% RSLogix 500 project DRYER MCM NOVEMBER NEW ZELAND 1-7-2018 CURRENT_JEFF_EMAIL_TO_EULISES.RSS, saved by version 11.00.00.00 %
PROJECT "ML1200"    % processor: MicroLogix 1200; MAIN_PROG %

PROGRAM FILES
  LAD 2 "MAIN_PROG"  11 rungs
  LAD 3 "DRYER CONT"  11 rungs
  LAD 4 "TEMPERATUR"  32 rungs
  LAD 5 "AIR PRES."  7 rungs
  LAD 6 "HUMIDITY"  13 rungs
  LAD 7 "RHL-TEMP"  2 rungs  % HEATING CONTROLS %
  LAD 8 "HEAT CONTR"  39 rungs
  LAD 9 "HOUR METER"  6 rungs
  LAD 10 "CONV CLEAN"  18 rungs  % Brush Cleaning %
  LAD 11 "FAULTS"  8 rungs

DATA FILES
  O0 OUTPUT  8 elements
  I1 INPUT  19 elements
  S2 STATUS  66 elements
  B3 BINARY  6 elements
  T4 TIMER  11 elements
  C5 COUNTER  1 elements
  R6 CONTROL  1 elements
  N7 INTEGER  80 elements
  F8 FLOAT  1 elements
  PD9 DRYER  4 elements

LADDER 2 "MAIN_PROG"
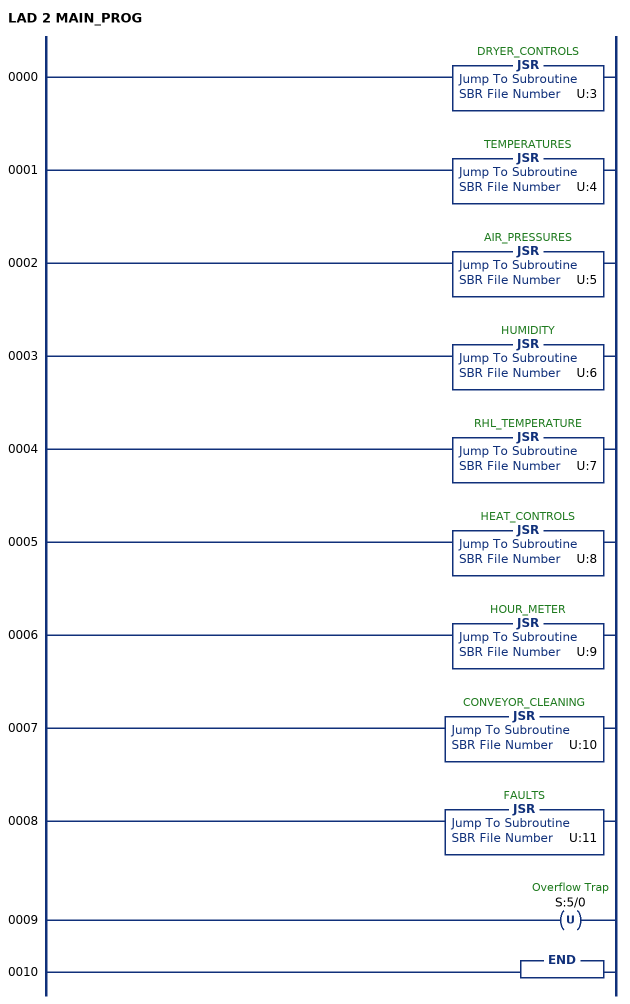
% Rung: 0 %
SOR JSR U:3 EOR
%   U:3  DRYER_CONTROLS %
% Rung: 1 %
SOR JSR U:4 EOR
%   U:4  TEMPERATURES %
% Rung: 2 %
SOR JSR U:5 EOR
%   U:5  AIR_PRESSURES %
% Rung: 3 %
SOR JSR U:6 EOR
%   U:6  HUMIDITY %
% Rung: 4 %
SOR JSR U:7 EOR
%   U:7  RHL_TEMPERATURE %
% Rung: 5 %
SOR JSR U:8 EOR
%   U:8  HEAT_CONTROLS %
% Rung: 6 %
SOR JSR U:9 EOR
%   U:9  HOUR_METER %
% Rung: 7 %
SOR JSR U:10 EOR
%   U:10  CONVEYOR_CLEANING %
% Rung: 8 %
SOR JSR U:11 EOR
%   U:11  FAULTS %
% Rung: 9 %
SOR OTU S:5/0 EOR
%   S:5/0  "Overflow Trap" %
% Rung: 10 %
SOR END EOR

LADDER 3 "DRYER CONT"
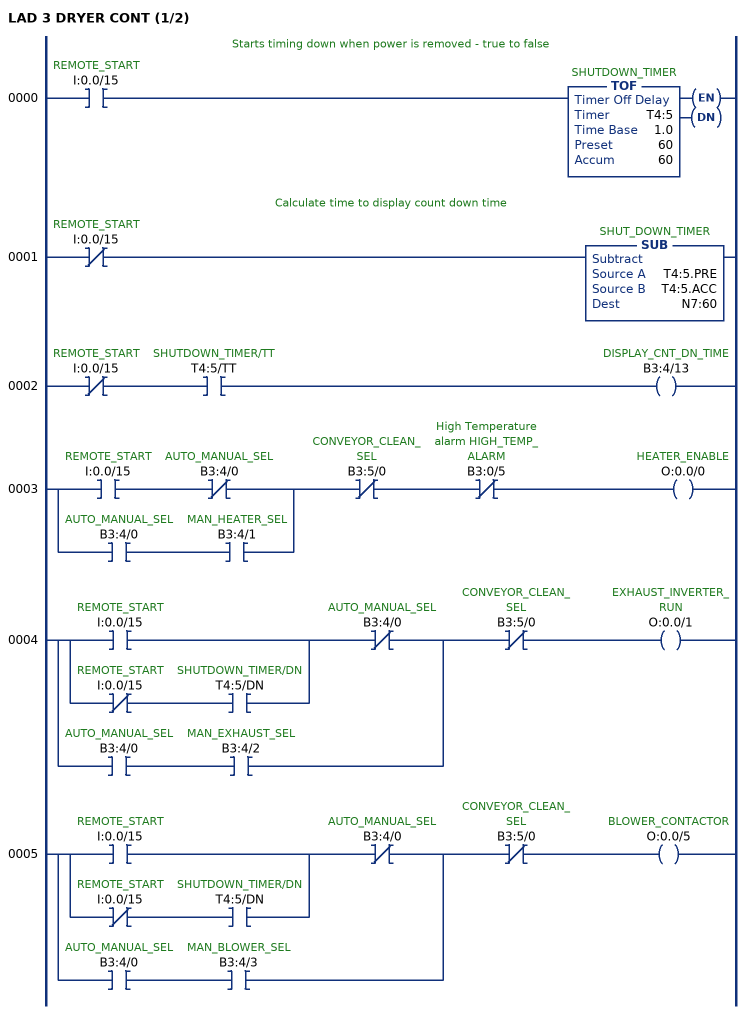
% Rung: 0 %
% Starts timing down when power is removed - true to false %
SOR XIC I:0.0/15 TOF T4:5 1.0 60 60 EOR
%   I:0.0/15  REMOTE_START %
%   T4:5  SHUTDOWN_TIMER %
% Rung: 1 %
% Calculate time to display count down time %
SOR XIO I:0.0/15 SUB T4:5.PRE T4:5.ACC N7:60 EOR
%   I:0.0/15  REMOTE_START %
%   T4:5  SHUTDOWN_TIMER %
%   N7:60  SHUT_DOWN_TIMER %
% Rung: 2 %
SOR XIO I:0.0/15 XIC T4:5/TT OTE B3:4/13 EOR
%   I:0.0/15  REMOTE_START %
%   T4:5  SHUTDOWN_TIMER %
%   B3:4/13  DISPLAY_CNT_DN_TIME %
% Rung: 3 %
SOR BST XIC I:0.0/15 XIO B3:4/0 NXB XIC B3:4/0 XIC B3:4/1 BND XIO B3:5/0 XIO B3:0/5 OTE O:0.0/0 EOR
%   I:0.0/15  REMOTE_START %
%   B3:4/0  AUTO_MANUAL_SEL %
%   B3:4/1  MAN_HEATER_SEL %
%   B3:5/0  CONVEYOR_CLEAN_SEL %
%   B3:0/5  HIGH_TEMP_ALARM  "High Temperature alarm" %
%   O:0.0/0  HEATER_ENABLE %
% Rung: 4 %
SOR BST BST XIC I:0.0/15 NXB XIO I:0.0/15 XIC T4:5/DN BND XIO B3:4/0 NXB XIC B3:4/0 XIC B3:4/2 BND XIO B3:5/0 OTE O:0.0/1 EOR
%   I:0.0/15  REMOTE_START %
%   T4:5  SHUTDOWN_TIMER %
%   B3:4/0  AUTO_MANUAL_SEL %
%   B3:4/2  MAN_EXHAUST_SEL %
%   B3:5/0  CONVEYOR_CLEAN_SEL %
%   O:0.0/1  EXHAUST_INVERTER_RUN %
% Rung: 5 %
SOR BST BST XIC I:0.0/15 NXB XIO I:0.0/15 XIC T4:5/DN BND XIO B3:4/0 NXB XIC B3:4/0 XIC B3:4/3 BND XIO B3:5/0 OTE O:0.0/5 EOR
%   I:0.0/15  REMOTE_START %
%   T4:5  SHUTDOWN_TIMER %
%   B3:4/0  AUTO_MANUAL_SEL %
%   B3:4/3  MAN_BLOWER_SEL %
%   B3:5/0  CONVEYOR_CLEAN_SEL %
%   O:0.0/5  BLOWER_CONTACTOR %

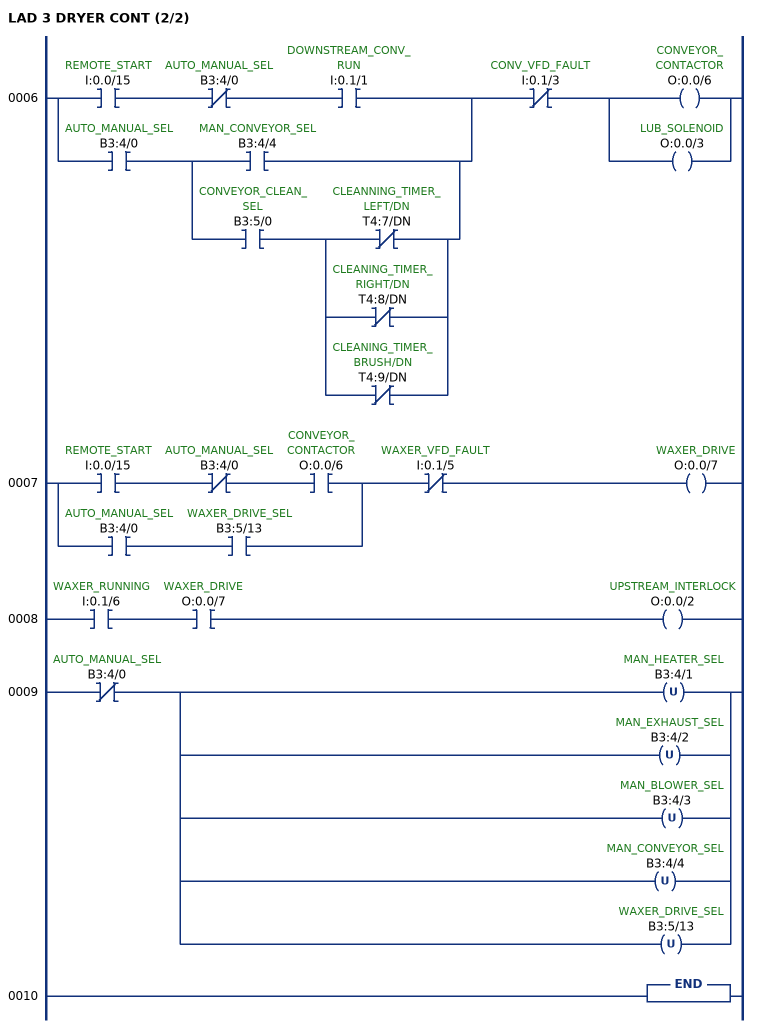
% Rung: 6 %
SOR BST XIC I:0.0/15 XIO B3:4/0 XIC I:0.1/1 NXB XIC B3:4/0 BST XIC B3:4/4 NXB XIC B3:5/0 BST XIO T4:7/DN NXB BST XIO T4:8/DN NXB XIO T4:9/DN BND BND BND BND XIO I:0.1/3 BST OTE O:0.0/6 NXB OTE O:0.0/3 BND EOR
%   I:0.0/15  REMOTE_START %
%   B3:4/0  AUTO_MANUAL_SEL %
%   I:0.1/1  DOWNSTREAM_CONV_RUN %
%   B3:4/4  MAN_CONVEYOR_SEL %
%   B3:5/0  CONVEYOR_CLEAN_SEL %
%   T4:7  CLEANNING_TIMER_LEFT %
%   T4:8  CLEANING_TIMER_RIGHT %
%   T4:9  CLEANING_TIMER_BRUSH %
%   I:0.1/3  CONV_VFD_FAULT %
%   O:0.0/6  CONVEYOR_CONTACTOR %
%   O:0.0/3  LUB_SOLENOID %
% Rung: 7 %
SOR BST XIC I:0.0/15 XIO B3:4/0 XIC O:0.0/6 NXB XIC B3:4/0 XIC B3:5/13 BND XIO I:0.1/5 OTE O:0.0/7 EOR
%   I:0.0/15  REMOTE_START %
%   B3:4/0  AUTO_MANUAL_SEL %
%   O:0.0/6  CONVEYOR_CONTACTOR %
%   B3:5/13  WAXER_DRIVE_SEL %
%   I:0.1/5  WAXER_VFD_FAULT %
%   O:0.0/7  WAXER_DRIVE %
% Rung: 8 %
SOR XIC I:0.1/6 XIC O:0.0/7 OTE O:0.0/2 EOR
%   I:0.1/6  WAXER_RUNNING %
%   O:0.0/7  WAXER_DRIVE %
%   O:0.0/2  UPSTREAM_INTERLOCK %
% Rung: 9 %
SOR XIO B3:4/0 BST BST BST BST OTU B3:4/1 NXB OTU B3:4/2 BND NXB OTU B3:4/3 BND NXB OTU B3:4/4 BND NXB OTU B3:5/13 BND EOR
%   B3:4/0  AUTO_MANUAL_SEL %
%   B3:4/1  MAN_HEATER_SEL %
%   B3:4/2  MAN_EXHAUST_SEL %
%   B3:4/3  MAN_BLOWER_SEL %
%   B3:4/4  MAN_CONVEYOR_SEL %
%   B3:5/13  WAXER_DRIVE_SEL %
% Rung: 10 %
SOR END EOR

LADDER 4 "TEMPERATUR"
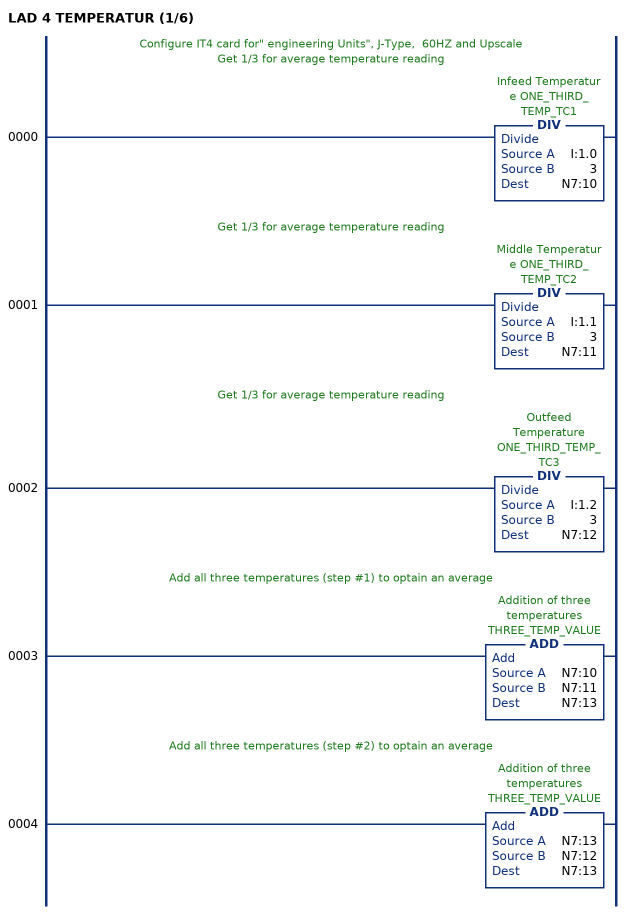
% Rung: 0 %
% Configure IT4 card for" engineering Units", J-Type,  60HZ and Upscale
% Get 1/3 for average temperature reading %
SOR DIV I:1.0 3 N7:10 EOR
%   I:1.0  INFEED_TEMP %
%   N7:10  ONE_THIRD_TEMP_TC1  "Infeed Temperature" %
% Rung: 1 %
% Get 1/3 for average temperature reading %
SOR DIV I:1.1 3 N7:11 EOR
%   I:1.1  MIDDLE_TEMP %
%   N7:11  ONE_THIRD_TEMP_TC2  "Middle Temperature" %
% Rung: 2 %
% Get 1/3 for average temperature reading %
SOR DIV I:1.2 3 N7:12 EOR
%   I:1.2  OUTFEED_TEMP %
%   N7:12  ONE_THIRD_TEMP_TC3  "Outfeed Temperature" %
% Rung: 3 %
% Add all three temperatures (step #1) to optain an average %
SOR ADD N7:10 N7:11 N7:13 EOR
%   N7:10  ONE_THIRD_TEMP_TC1  "Infeed Temperature" %
%   N7:11  ONE_THIRD_TEMP_TC2  "Middle Temperature" %
%   N7:13  THREE_TEMP_VALUE  "Addition of three temperatures" %
% Rung: 4 %
% Add all three temperatures (step #2) to optain an average %
SOR ADD N7:13 N7:12 N7:13 EOR
%   N7:13  THREE_TEMP_VALUE  "Addition of three temperatures" %
%   N7:12  ONE_THIRD_TEMP_TC3  "Outfeed Temperature" %

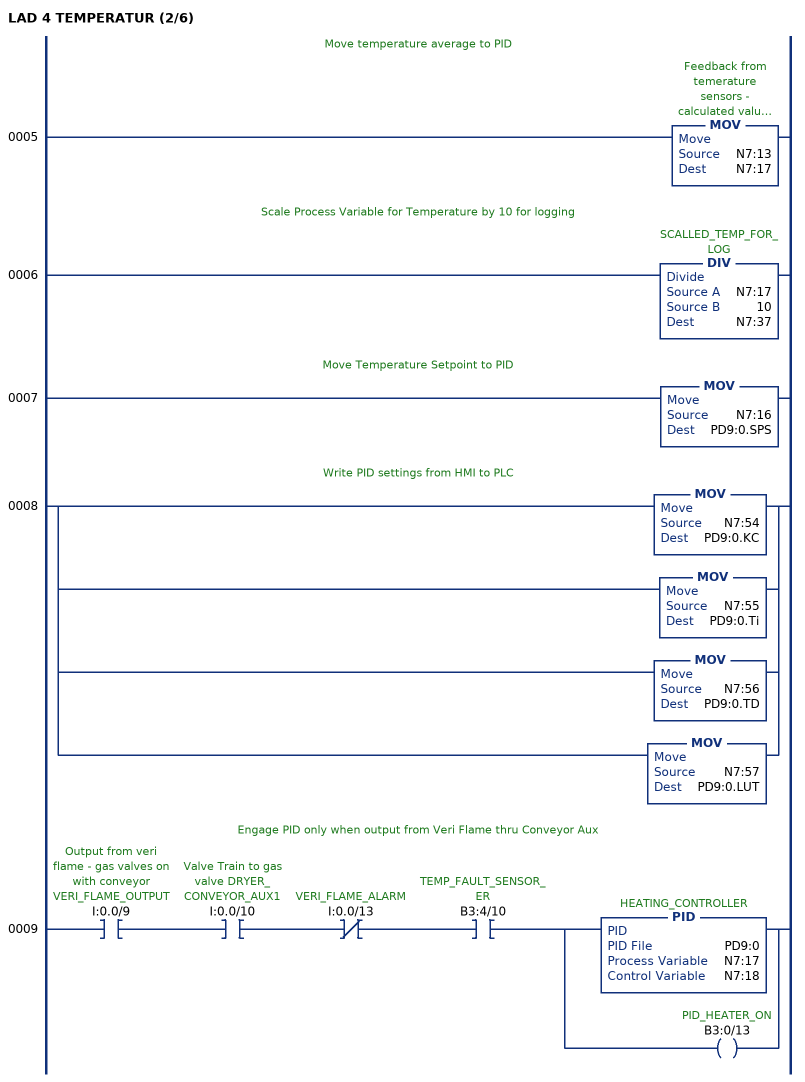
% Rung: 5 %
% Move temperature average to PID %
SOR MOV N7:13 N7:17 EOR
%   N7:13  THREE_TEMP_VALUE  "Addition of three temperatures" %
%   N7:17  PV_TEMP_PROCESS_VAR  "Feedback from temerature sensors - calculated value" %
% Rung: 6 %
% Scale Process Variable for Temperature by 10 for logging %
SOR DIV N7:17 10 N7:37 EOR
%   N7:17  PV_TEMP_PROCESS_VAR  "Feedback from temerature sensors - calculated value" %
%   N7:37  SCALLED_TEMP_FOR_LOG %
% Rung: 7 %
% Move Temperature Setpoint to PID %
SOR MOV N7:16 PD9:0.SPS EOR
%   N7:16  SPS_TEMP_SETPOINT  "Display Input Value - desired Temperature" %
% Rung: 8 %
% Write PID settings from HMI to PLC %
SOR BST BST BST MOV N7:54 PD9:0.KC NXB MOV N7:55 PD9:0.Ti BND NXB MOV N7:56 PD9:0.TD BND NXB MOV N7:57 PD9:0.LUT BND EOR
%   N7:54  PID_KC %
%   N7:55  PID_TI %
%   N7:56  PID_TD %
%   N7:57  PID_LUT %
% Rung: 9 %
% Engage PID only when output from Veri Flame thru Conveyor Aux %
SOR XIC I:0.0/9 XIC I:0.0/10 XIO I:0.0/13 XIC B3:4/10 BST PID PD9:0 N7:17 N7:18 NXB OTE B3:0/13 BND EOR
%   I:0.0/9  VERI_FLAME_OUTPUT  "Output from veri flame - gas valves on with conveyor" %
%   I:0.0/10  DRYER_CONVEYOR_AUX1  "Valve Train to gas valve" %
%   I:0.0/13  VERI_FLAME_ALARM %
%   B3:4/10  TEMP_FAULT_SENSOR_ER %
%   PD9:0  HEATING_CONTROLLER %
%   N7:17  PV_TEMP_PROCESS_VAR  "Feedback from temerature sensors - calculated value" %
%   N7:18  CV_TEMP_CONTROL_VAR  "Output value to output for output card" %
%   B3:0/13  PID_HEATER_ON %

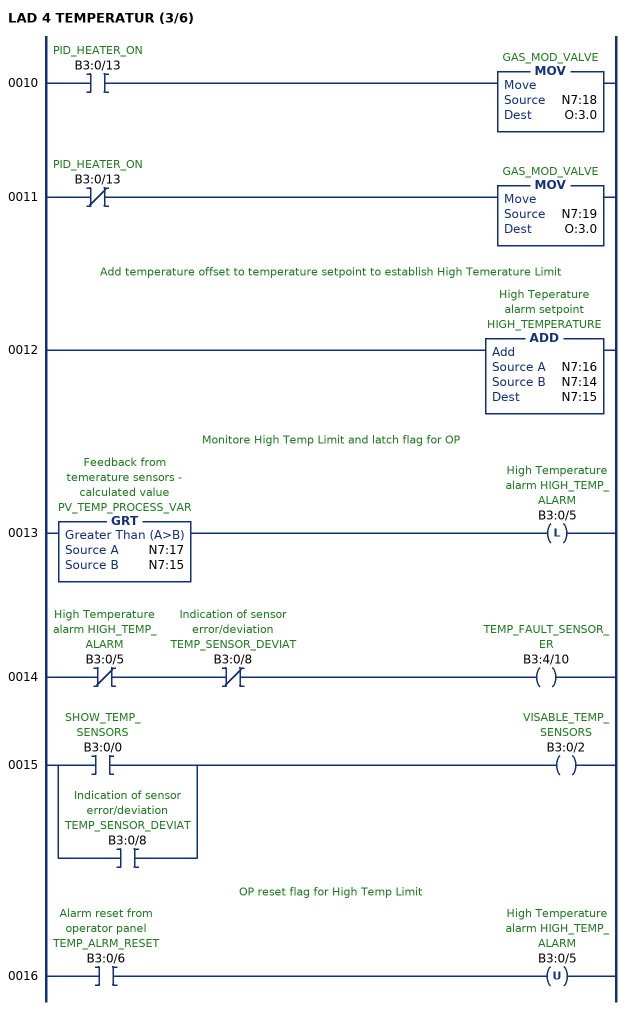
% Rung: 10 %
SOR XIC B3:0/13 MOV N7:18 O:3.0 EOR
%   B3:0/13  PID_HEATER_ON %
%   N7:18  CV_TEMP_CONTROL_VAR  "Output value to output for output card" %
%   O:3.0  GAS_MOD_VALVE %
% Rung: 11 %
SOR XIO B3:0/13 MOV N7:19 O:3.0 EOR
%   B3:0/13  PID_HEATER_ON %
%   N7:19  MIN_GAS_VALVE_POS  "When Conveyor Aux is off, throttle valve back" %
%   O:3.0  GAS_MOD_VALVE %
% Rung: 12 %
% Add temperature offset to temperature setpoint to establish High Temerature Limit %
SOR ADD N7:16 N7:14 N7:15 EOR
%   N7:16  SPS_TEMP_SETPOINT  "Display Input Value - desired Temperature" %
%   N7:14  HIGH_TEMP_OFFSET  "Value added to Temp Setpoint to set high temerature" %
%   N7:15  HIGH_TEMPERATURE  "High Teperature alarm setpoint" %
% Rung: 13 %
% Monitore High Temp Limit and latch flag for OP %
SOR GRT N7:17 N7:15 OTL B3:0/5 EOR
%   N7:17  PV_TEMP_PROCESS_VAR  "Feedback from temerature sensors - calculated value" %
%   N7:15  HIGH_TEMPERATURE  "High Teperature alarm setpoint" %
%   B3:0/5  HIGH_TEMP_ALARM  "High Temperature alarm" %
% Rung: 14 %
SOR XIO B3:0/5 XIO B3:0/8 OTE B3:4/10 EOR
%   B3:0/5  HIGH_TEMP_ALARM  "High Temperature alarm" %
%   B3:0/8  TEMP_SENSOR_DEVIAT  "Indication of sensor error/deviation" %
%   B3:4/10  TEMP_FAULT_SENSOR_ER %
% Rung: 15 %
SOR BST XIC B3:0/0 NXB XIC B3:0/8 BND OTE B3:0/2 EOR
%   B3:0/0  SHOW_TEMP_SENSORS %
%   B3:0/8  TEMP_SENSOR_DEVIAT  "Indication of sensor error/deviation" %
%   B3:0/2  VISABLE_TEMP_SENSORS %
% Rung: 16 %
% OP reset flag for High Temp Limit %
SOR XIC B3:0/6 OTU B3:0/5 EOR
%   B3:0/6  TEMP_ALRM_RESET  "Alarm reset from operator panel" %
%   B3:0/5  HIGH_TEMP_ALARM  "High Temperature alarm" %

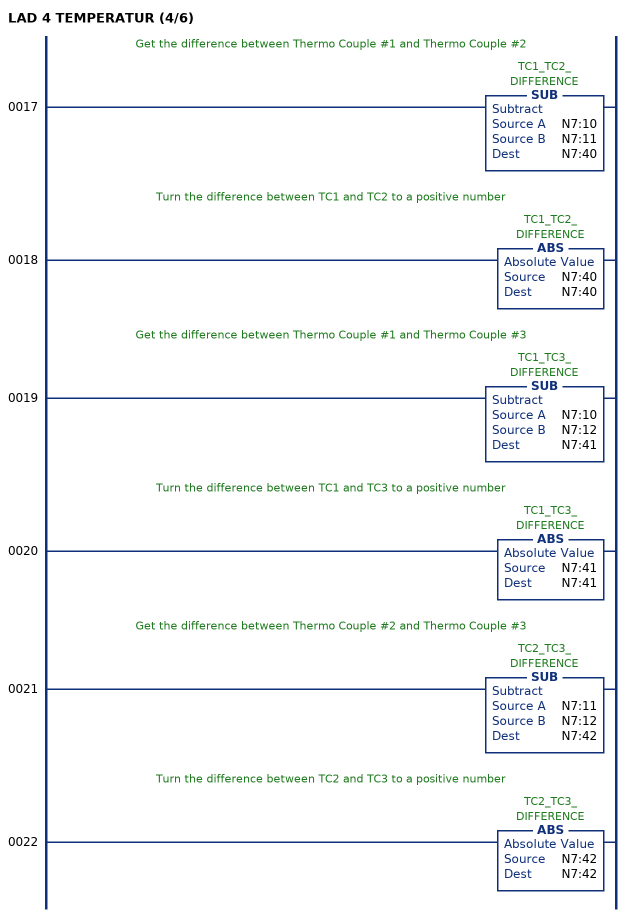
% Rung: 17 %
% Get the difference between Thermo Couple #1 and Thermo Couple #2 %
SOR SUB N7:10 N7:11 N7:40 EOR
%   N7:10  ONE_THIRD_TEMP_TC1  "Infeed Temperature" %
%   N7:11  ONE_THIRD_TEMP_TC2  "Middle Temperature" %
%   N7:40  TC1_TC2_DIFFERENCE %
% Rung: 18 %
% Turn the difference between TC1 and TC2 to a positive number %
SOR ABS N7:40 N7:40 EOR
%   N7:40  TC1_TC2_DIFFERENCE %
% Rung: 19 %
% Get the difference between Thermo Couple #1 and Thermo Couple #3 %
SOR SUB N7:10 N7:12 N7:41 EOR
%   N7:10  ONE_THIRD_TEMP_TC1  "Infeed Temperature" %
%   N7:12  ONE_THIRD_TEMP_TC3  "Outfeed Temperature" %
%   N7:41  TC1_TC3_DIFFERENCE %
% Rung: 20 %
% Turn the difference between TC1 and TC3 to a positive number %
SOR ABS N7:41 N7:41 EOR
%   N7:41  TC1_TC3_DIFFERENCE %
% Rung: 21 %
% Get the difference between Thermo Couple #2 and Thermo Couple #3 %
SOR SUB N7:11 N7:12 N7:42 EOR
%   N7:11  ONE_THIRD_TEMP_TC2  "Middle Temperature" %
%   N7:12  ONE_THIRD_TEMP_TC3  "Outfeed Temperature" %
%   N7:42  TC2_TC3_DIFFERENCE %
% Rung: 22 %
% Turn the difference between TC2 and TC3 to a positive number %
SOR ABS N7:42 N7:42 EOR
%   N7:42  TC2_TC3_DIFFERENCE %

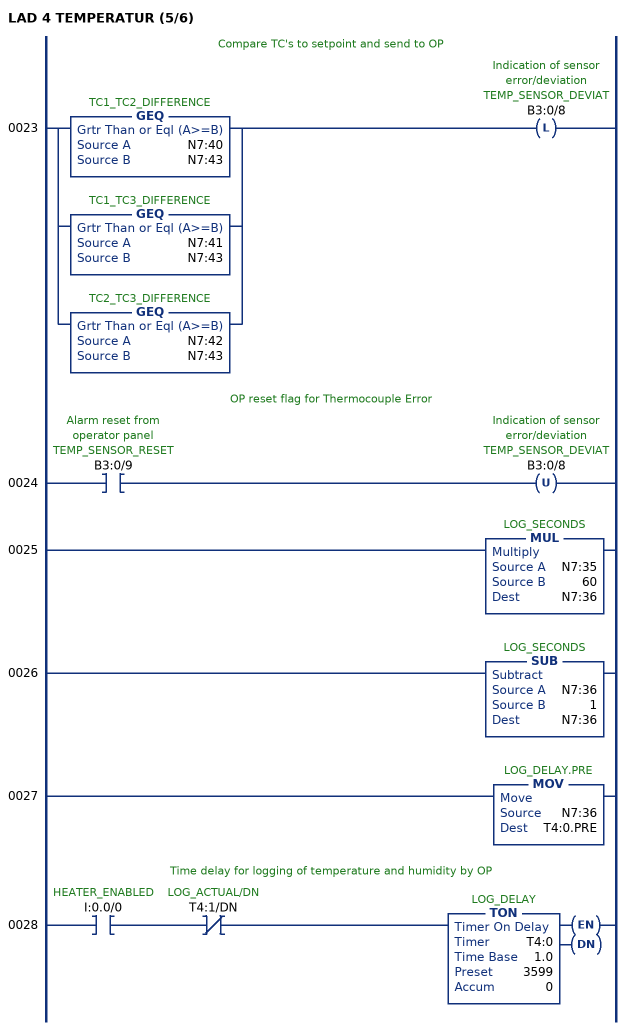
% Rung: 23 %
% Compare TC's to setpoint and send to OP %
SOR BST GEQ N7:40 N7:43 NXB BST GEQ N7:41 N7:43 NXB GEQ N7:42 N7:43 BND BND OTL B3:0/8 EOR
%   N7:40  TC1_TC2_DIFFERENCE %
%   N7:43  MAX_TEMP_SENSOR_DEV %
%   N7:41  TC1_TC3_DIFFERENCE %
%   N7:42  TC2_TC3_DIFFERENCE %
%   B3:0/8  TEMP_SENSOR_DEVIAT  "Indication of sensor error/deviation" %
% Rung: 24 %
% OP reset flag for Thermocouple Error %
SOR XIC B3:0/9 OTU B3:0/8 EOR
%   B3:0/9  TEMP_SENSOR_RESET  "Alarm reset from operator panel" %
%   B3:0/8  TEMP_SENSOR_DEVIAT  "Indication of sensor error/deviation" %
% Rung: 25 %
SOR MUL N7:35 60 N7:36 EOR
%   N7:35  LOG_MINUTES %
%   N7:36  LOG_SECONDS %
% Rung: 26 %
SOR SUB N7:36 1 N7:36 EOR
%   N7:36  LOG_SECONDS %
% Rung: 27 %
SOR MOV N7:36 T4:0.PRE EOR
%   N7:36  LOG_SECONDS %
%   T4:0  LOG_DELAY %
% Rung: 28 %
% Time delay for logging of temperature and humidity by OP %
SOR XIC I:0.0/0 XIO T4:1/DN TON T4:0 1.0 3599 0 EOR
%   I:0.0/0  HEATER_ENABLED %
%   T4:1  LOG_ACTUAL %
%   T4:0  LOG_DELAY %

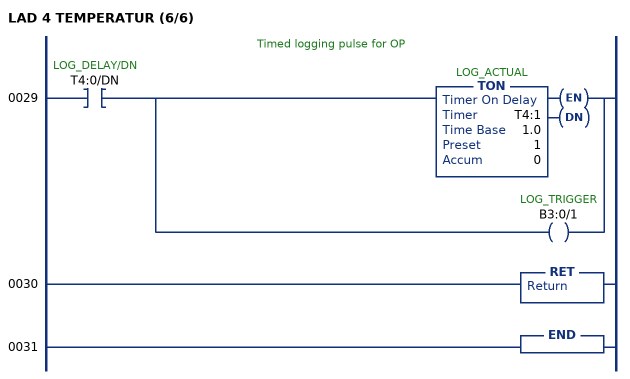
% Rung: 29 %
% Timed logging pulse for OP %
SOR XIC T4:0/DN BST TON T4:1 1.0 1 0 NXB OTE B3:0/1 BND EOR
%   T4:0  LOG_DELAY %
%   T4:1  LOG_ACTUAL %
%   B3:0/1  LOG_TRIGGER %
% Rung: 30 %
SOR RET EOR
% Rung: 31 %
SOR END EOR

LADDER 5 "AIR PRES."
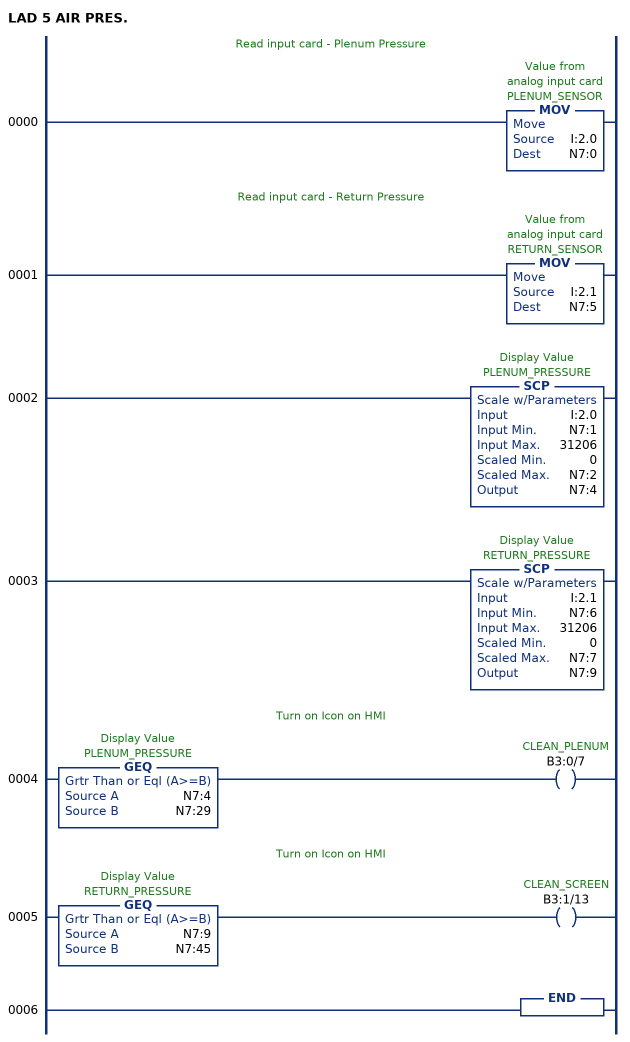
% Rung: 0 %
% Read input card - Plenum Pressure %
SOR MOV I:2.0 N7:0 EOR
%   N7:0  PLENUM_SENSOR  "Value from analog input card" %
% Rung: 1 %
% Read input card - Return Pressure %
SOR MOV I:2.1 N7:5 EOR
%   N7:5  RETURN_SENSOR  "Value from analog input card" %
% Rung: 2 %
SOR SCP I:2.0 N7:1 31206 0 N7:2 N7:4 EOR
%   N7:1  PLENUM_ZERO  "The amount needed to return a zero value with no pressure" %
%   N7:2  PLENUM_SCALLING_MAX  "Max range of sensor" %
%   N7:4  PLENUM_PRESSURE  "Display Value" %
% Rung: 3 %
SOR SCP I:2.1 N7:6 31206 0 N7:7 N7:9 EOR
%   N7:6  RETURN_ZERO  "The amount needed to return a zero value with no pressure" %
%   N7:7  RETURN_SCALING_MAX  "Max range of sensor" %
%   N7:9  RETURN_PRESSURE  "Display Value" %
% Rung: 4 %
% Turn on Icon on HMI %
SOR GEQ N7:4 N7:29 OTE B3:0/7 EOR
%   N7:4  PLENUM_PRESSURE  "Display Value" %
%   N7:29  PLENUM_ALARM  "signal Operator Panel that cleaning is required" %
%   B3:0/7  CLEAN_PLENUM %
% Rung: 5 %
% Turn on Icon on HMI %
SOR GEQ N7:9 N7:45 OTE B3:1/13 EOR
%   N7:9  RETURN_PRESSURE  "Display Value" %
%   N7:45  CLEAN_SCREEN_ALARM %
%   B3:1/13  CLEAN_SCREEN %
% Rung: 6 %
SOR END EOR

LADDER 6 "HUMIDITY"
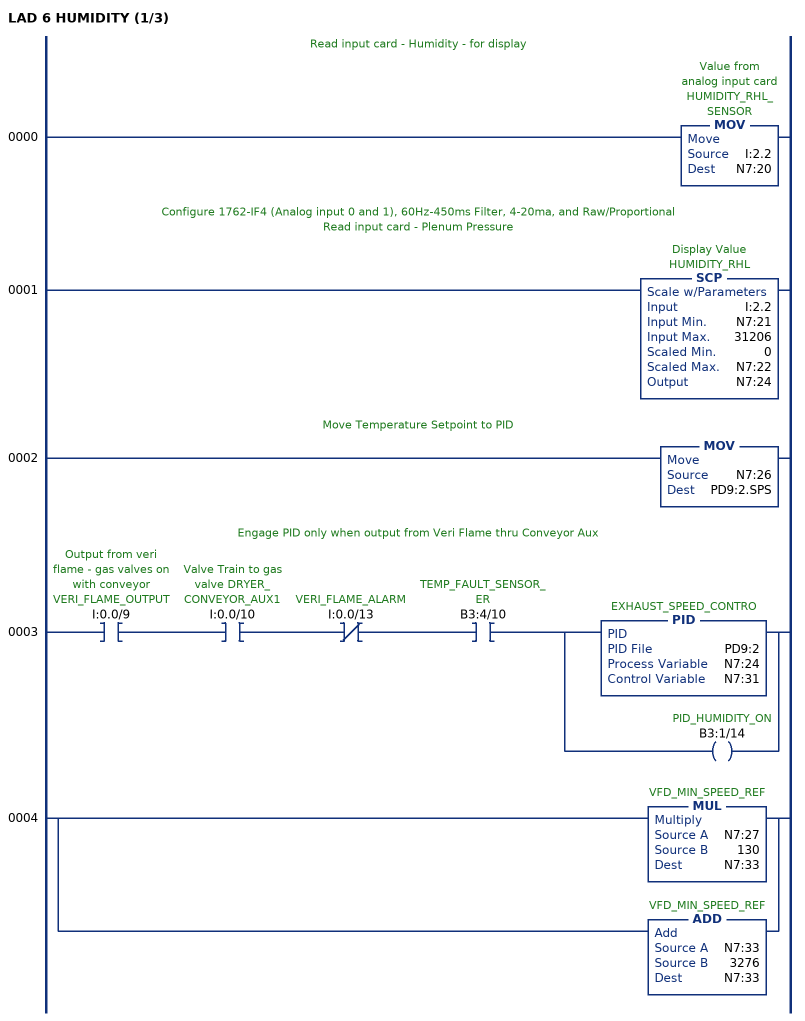
% Rung: 0 %
% Read input card - Humidity - for display %
SOR MOV I:2.2 N7:20 EOR
%   N7:20  HUMIDITY_RHL_SENSOR  "Value from analog input card" %
% Rung: 1 %
% Configure 1762-IF4 (Analog input 0 and 1), 60Hz-450ms Filter, 4-20ma, and Raw/Proportional
% Read input card - Plenum Pressure %
SOR SCP I:2.2 N7:21 31206 0 N7:22 N7:24 EOR
%   N7:21  HUMIDITY_ZERO  "The amount needed to return a zero value with no humitity" %
%   N7:22  HUMIDITY_SCALING_MAX  "Max range of sensor" %
%   N7:24  HUMIDITY_RHL  "Display Value" %
% Rung: 2 %
% Move Temperature Setpoint to PID %
SOR MOV N7:26 PD9:2.SPS EOR
%   N7:26  HUMITITY_MAX_SETPOIN %
% Rung: 3 %
% Engage PID only when output from Veri Flame thru Conveyor Aux %
SOR XIC I:0.0/9 XIC I:0.0/10 XIO I:0.0/13 XIC B3:4/10 BST PID PD9:2 N7:24 N7:31 NXB OTE B3:1/14 BND EOR
%   I:0.0/9  VERI_FLAME_OUTPUT  "Output from veri flame - gas valves on with conveyor" %
%   I:0.0/10  DRYER_CONVEYOR_AUX1  "Valve Train to gas valve" %
%   I:0.0/13  VERI_FLAME_ALARM %
%   B3:4/10  TEMP_FAULT_SENSOR_ER %
%   PD9:2  EXHAUST_SPEED_CONTRO %
%   N7:24  HUMIDITY_RHL  "Display Value" %
%   N7:31  CV_RH_CONTROL_VAR  "Output value to output for output card" %
%   B3:1/14  PID_HUMIDITY_ON %
% Rung: 4 %
SOR BST MUL N7:27 130 N7:33 NXB ADD N7:33 3276 N7:33 BND EOR
%   N7:27  EXHAUST_MIN_SPEED %
%   N7:33  VFD_MIN_SPEED_REF %

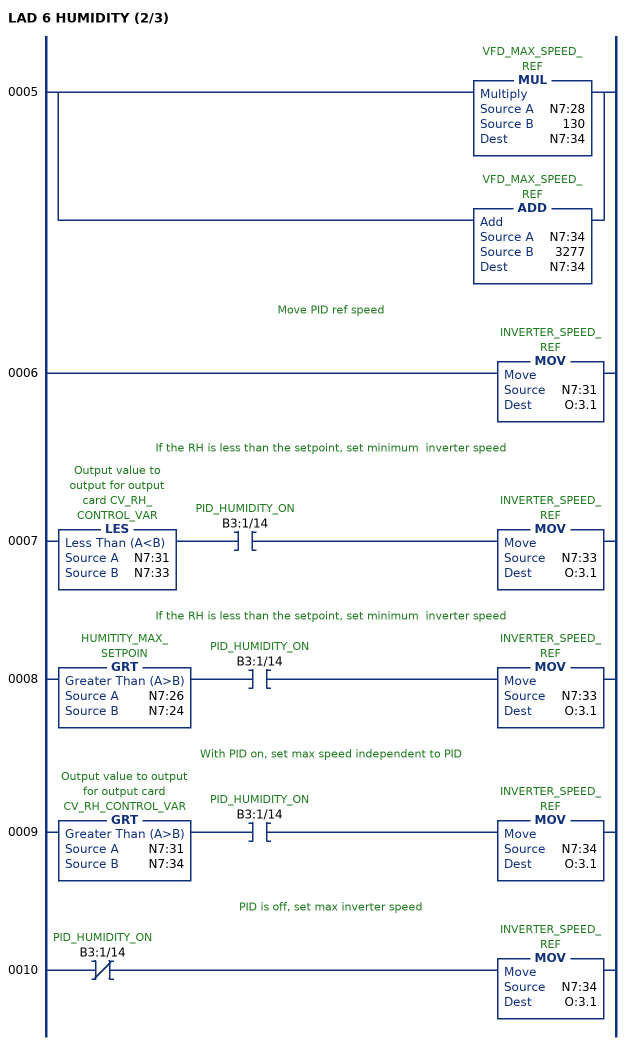
% Rung: 5 %
SOR BST MUL N7:28 130 N7:34 NXB ADD N7:34 3277 N7:34 BND EOR
%   N7:28  EXHAUST_MAX_SPEED %
%   N7:34  VFD_MAX_SPEED_REF %
% Rung: 6 %
% Move PID ref speed %
SOR MOV N7:31 O:3.1 EOR
%   N7:31  CV_RH_CONTROL_VAR  "Output value to output for output card" %
%   O:3.1  INVERTER_SPEED_REF %
% Rung: 7 %
% If the RH is less than the setpoint, set minimum  inverter speed %
SOR LES N7:31 N7:33 XIC B3:1/14 MOV N7:33 O:3.1 EOR
%   N7:31  CV_RH_CONTROL_VAR  "Output value to output for output card" %
%   N7:33  VFD_MIN_SPEED_REF %
%   B3:1/14  PID_HUMIDITY_ON %
%   O:3.1  INVERTER_SPEED_REF %
% Rung: 8 %
% If the RH is less than the setpoint, set minimum  inverter speed %
SOR GRT N7:26 N7:24 XIC B3:1/14 MOV N7:33 O:3.1 EOR
%   N7:26  HUMITITY_MAX_SETPOIN %
%   N7:24  HUMIDITY_RHL  "Display Value" %
%   B3:1/14  PID_HUMIDITY_ON %
%   N7:33  VFD_MIN_SPEED_REF %
%   O:3.1  INVERTER_SPEED_REF %
% Rung: 9 %
% With PID on, set max speed independent to PID %
SOR GRT N7:31 N7:34 XIC B3:1/14 MOV N7:34 O:3.1 EOR
%   N7:31  CV_RH_CONTROL_VAR  "Output value to output for output card" %
%   N7:34  VFD_MAX_SPEED_REF %
%   B3:1/14  PID_HUMIDITY_ON %
%   O:3.1  INVERTER_SPEED_REF %
% Rung: 10 %
% PID is off, set max inverter speed %
SOR XIO B3:1/14 MOV N7:34 O:3.1 EOR
%   B3:1/14  PID_HUMIDITY_ON %
%   N7:34  VFD_MAX_SPEED_REF %
%   O:3.1  INVERTER_SPEED_REF %

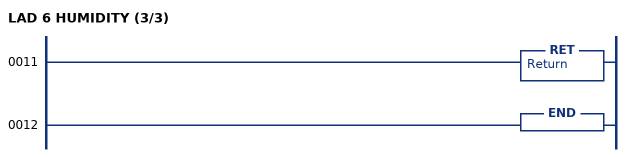
% Rung: 11 %
SOR RET EOR
% Rung: 12 %
SOR END EOR

LADDER 7 "RHL-TEMP"    % HEATING CONTROLS %
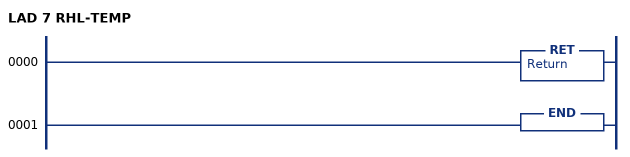
% Rung: 0 %
SOR RET EOR
% Rung: 1 %
SOR END EOR

LADDER 8 "HEAT CONTR"
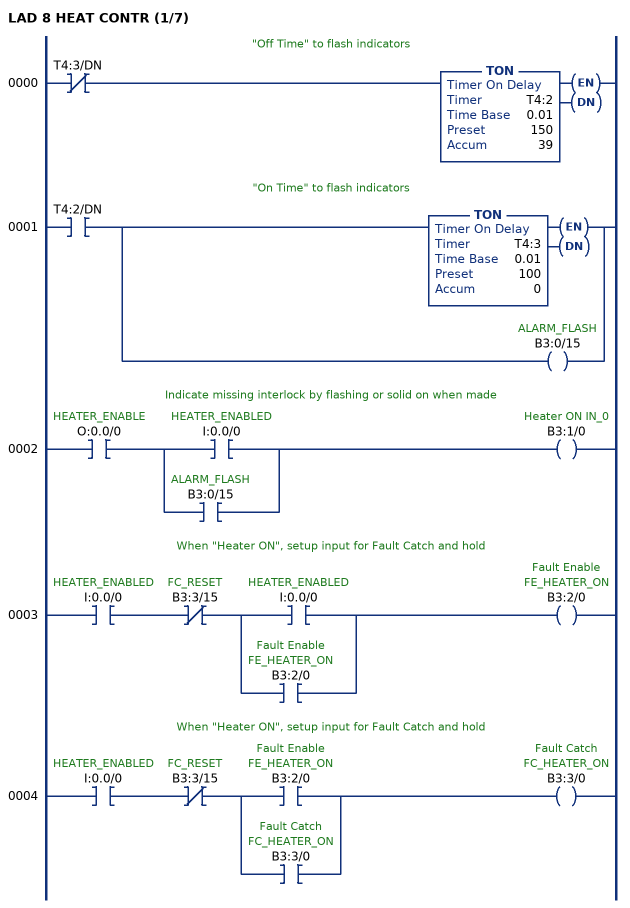
% Rung: 0 %
% "Off Time" to flash indicators %
SOR XIO T4:3/DN TON T4:2 0.01 150 39 EOR
% Rung: 1 %
% "On Time" to flash indicators %
SOR XIC T4:2/DN BST TON T4:3 0.01 100 0 NXB OTE B3:0/15 BND EOR
%   B3:0/15  ALARM_FLASH %
% Rung: 2 %
% Indicate missing interlock by flashing or solid on when made %
SOR XIC O:0.0/0 BST XIC I:0.0/0 NXB XIC B3:0/15 BND OTE B3:1/0 EOR
%   O:0.0/0  HEATER_ENABLE %
%   I:0.0/0  HEATER_ENABLED %
%   B3:0/15  ALARM_FLASH %
%   B3:1/0  IN_0  "Heater ON" %
% Rung: 3 %
% When "Heater ON", setup input for Fault Catch and hold %
SOR XIC I:0.0/0 XIO B3:3/15 BST XIC I:0.0/0 NXB XIC B3:2/0 BND OTE B3:2/0 EOR
%   I:0.0/0  HEATER_ENABLED %
%   B3:3/15  FC_RESET %
%   B3:2/0  FE_HEATER_ON  "Fault Enable" %
% Rung: 4 %
% When "Heater ON", setup input for Fault Catch and hold %
SOR XIC I:0.0/0 XIO B3:3/15 BST XIC B3:2/0 NXB XIC B3:3/0 BND OTE B3:3/0 EOR
%   I:0.0/0  HEATER_ENABLED %
%   B3:3/15  FC_RESET %
%   B3:2/0  FE_HEATER_ON  "Fault Enable" %
%   B3:3/0  FC_HEATER_ON  "Fault Catch" %

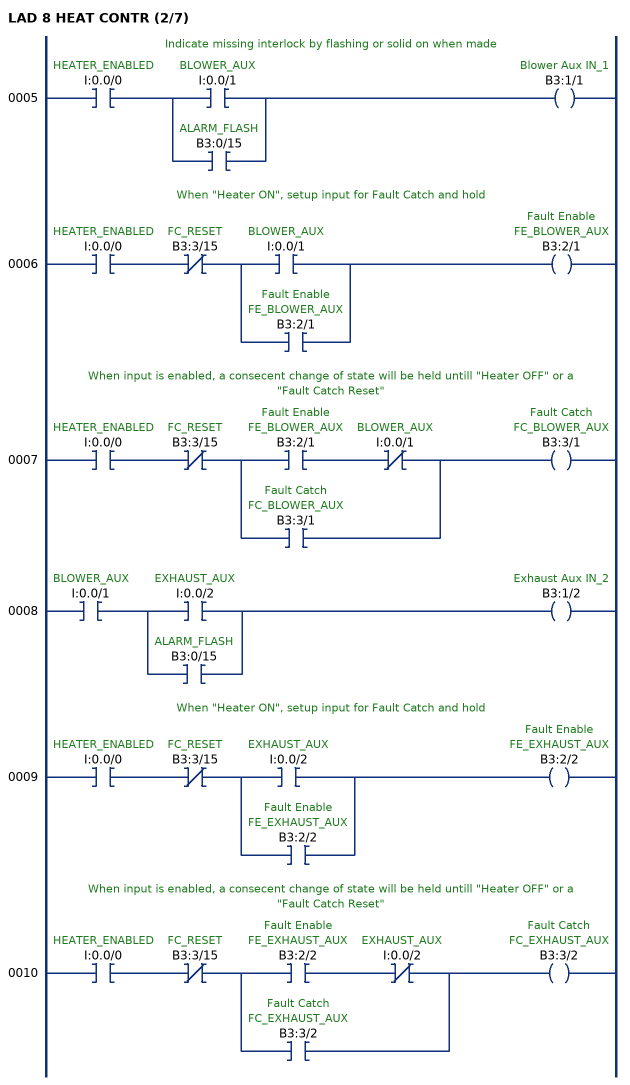
% Rung: 5 %
% Indicate missing interlock by flashing or solid on when made %
SOR XIC I:0.0/0 BST XIC I:0.0/1 NXB XIC B3:0/15 BND OTE B3:1/1 EOR
%   I:0.0/0  HEATER_ENABLED %
%   I:0.0/1  BLOWER_AUX %
%   B3:0/15  ALARM_FLASH %
%   B3:1/1  IN_1  "Blower Aux" %
% Rung: 6 %
% When "Heater ON", setup input for Fault Catch and hold %
SOR XIC I:0.0/0 XIO B3:3/15 BST XIC I:0.0/1 NXB XIC B3:2/1 BND OTE B3:2/1 EOR
%   I:0.0/0  HEATER_ENABLED %
%   B3:3/15  FC_RESET %
%   I:0.0/1  BLOWER_AUX %
%   B3:2/1  FE_BLOWER_AUX  "Fault Enable" %
% Rung: 7 %
% When input is enabled, a consecent change of state will be held untill "Heater OFF" or a "Fault Catch Reset" %
SOR XIC I:0.0/0 XIO B3:3/15 BST XIC B3:2/1 XIO I:0.0/1 NXB XIC B3:3/1 BND OTE B3:3/1 EOR
%   I:0.0/0  HEATER_ENABLED %
%   B3:3/15  FC_RESET %
%   B3:2/1  FE_BLOWER_AUX  "Fault Enable" %
%   I:0.0/1  BLOWER_AUX %
%   B3:3/1  FC_BLOWER_AUX  "Fault Catch" %
% Rung: 8 %
SOR XIC I:0.0/1 BST XIC I:0.0/2 NXB XIC B3:0/15 BND OTE B3:1/2 EOR
%   I:0.0/1  BLOWER_AUX %
%   I:0.0/2  EXHAUST_AUX %
%   B3:0/15  ALARM_FLASH %
%   B3:1/2  IN_2  "Exhaust Aux" %
% Rung: 9 %
% When "Heater ON", setup input for Fault Catch and hold %
SOR XIC I:0.0/0 XIO B3:3/15 BST XIC I:0.0/2 NXB XIC B3:2/2 BND OTE B3:2/2 EOR
%   I:0.0/0  HEATER_ENABLED %
%   B3:3/15  FC_RESET %
%   I:0.0/2  EXHAUST_AUX %
%   B3:2/2  FE_EXHAUST_AUX  "Fault Enable" %
% Rung: 10 %
% When input is enabled, a consecent change of state will be held untill "Heater OFF" or a "Fault Catch Reset" %
SOR XIC I:0.0/0 XIO B3:3/15 BST XIC B3:2/2 XIO I:0.0/2 NXB XIC B3:3/2 BND OTE B3:3/2 EOR
%   I:0.0/0  HEATER_ENABLED %
%   B3:3/15  FC_RESET %
%   B3:2/2  FE_EXHAUST_AUX  "Fault Enable" %
%   I:0.0/2  EXHAUST_AUX %
%   B3:3/2  FC_EXHAUST_AUX  "Fault Catch" %

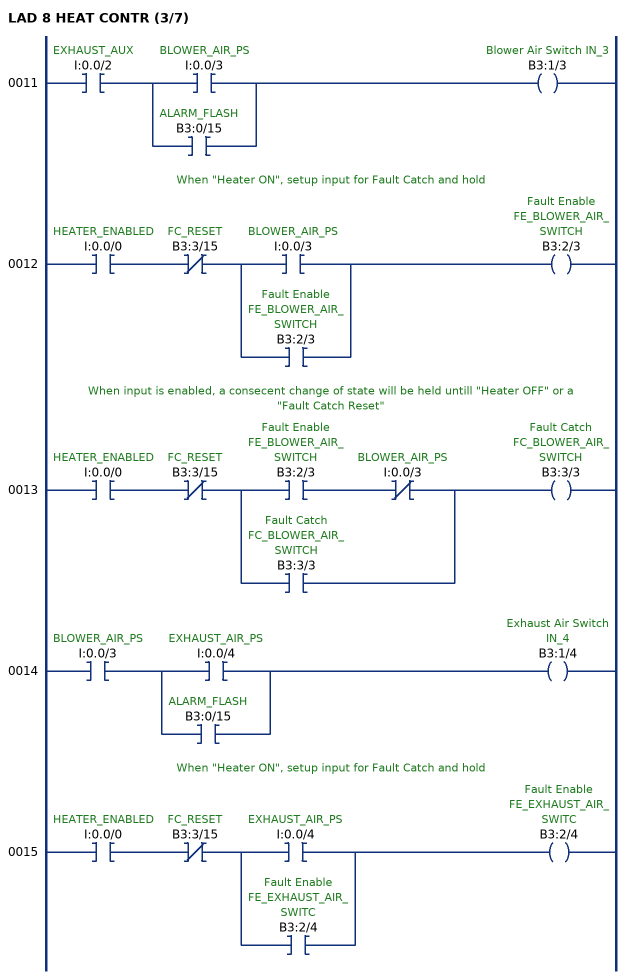
% Rung: 11 %
SOR XIC I:0.0/2 BST XIC I:0.0/3 NXB XIC B3:0/15 BND OTE B3:1/3 EOR
%   I:0.0/2  EXHAUST_AUX %
%   I:0.0/3  BLOWER_AIR_PS %
%   B3:0/15  ALARM_FLASH %
%   B3:1/3  IN_3  "Blower Air Switch" %
% Rung: 12 %
% When "Heater ON", setup input for Fault Catch and hold %
SOR XIC I:0.0/0 XIO B3:3/15 BST XIC I:0.0/3 NXB XIC B3:2/3 BND OTE B3:2/3 EOR
%   I:0.0/0  HEATER_ENABLED %
%   B3:3/15  FC_RESET %
%   I:0.0/3  BLOWER_AIR_PS %
%   B3:2/3  FE_BLOWER_AIR_SWITCH  "Fault Enable" %
% Rung: 13 %
% When input is enabled, a consecent change of state will be held untill "Heater OFF" or a "Fault Catch Reset" %
SOR XIC I:0.0/0 XIO B3:3/15 BST XIC B3:2/3 XIO I:0.0/3 NXB XIC B3:3/3 BND OTE B3:3/3 EOR
%   I:0.0/0  HEATER_ENABLED %
%   B3:3/15  FC_RESET %
%   B3:2/3  FE_BLOWER_AIR_SWITCH  "Fault Enable" %
%   I:0.0/3  BLOWER_AIR_PS %
%   B3:3/3  FC_BLOWER_AIR_SWITCH  "Fault Catch" %
% Rung: 14 %
SOR XIC I:0.0/3 BST XIC I:0.0/4 NXB XIC B3:0/15 BND OTE B3:1/4 EOR
%   I:0.0/3  BLOWER_AIR_PS %
%   I:0.0/4  EXHAUST_AIR_PS %
%   B3:0/15  ALARM_FLASH %
%   B3:1/4  IN_4  "Exhaust Air Switch" %
% Rung: 15 %
% When "Heater ON", setup input for Fault Catch and hold %
SOR XIC I:0.0/0 XIO B3:3/15 BST XIC I:0.0/4 NXB XIC B3:2/4 BND OTE B3:2/4 EOR
%   I:0.0/0  HEATER_ENABLED %
%   B3:3/15  FC_RESET %
%   I:0.0/4  EXHAUST_AIR_PS %
%   B3:2/4  FE_EXHAUST_AIR_SWITC  "Fault Enable" %

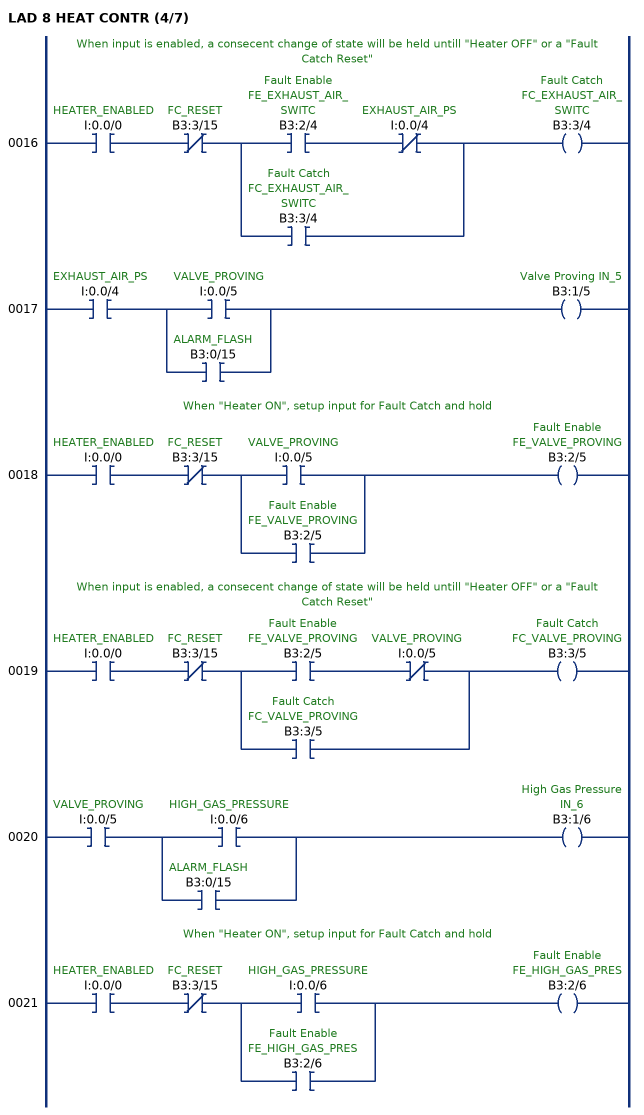
% Rung: 16 %
% When input is enabled, a consecent change of state will be held untill "Heater OFF" or a "Fault Catch Reset" %
SOR XIC I:0.0/0 XIO B3:3/15 BST XIC B3:2/4 XIO I:0.0/4 NXB XIC B3:3/4 BND OTE B3:3/4 EOR
%   I:0.0/0  HEATER_ENABLED %
%   B3:3/15  FC_RESET %
%   B3:2/4  FE_EXHAUST_AIR_SWITC  "Fault Enable" %
%   I:0.0/4  EXHAUST_AIR_PS %
%   B3:3/4  FC_EXHAUST_AIR_SWITC  "Fault Catch" %
% Rung: 17 %
SOR XIC I:0.0/4 BST XIC I:0.0/5 NXB XIC B3:0/15 BND OTE B3:1/5 EOR
%   I:0.0/4  EXHAUST_AIR_PS %
%   I:0.0/5  VALVE_PROVING %
%   B3:0/15  ALARM_FLASH %
%   B3:1/5  IN_5  "Valve Proving" %
% Rung: 18 %
% When "Heater ON", setup input for Fault Catch and hold %
SOR XIC I:0.0/0 XIO B3:3/15 BST XIC I:0.0/5 NXB XIC B3:2/5 BND OTE B3:2/5 EOR
%   I:0.0/0  HEATER_ENABLED %
%   B3:3/15  FC_RESET %
%   I:0.0/5  VALVE_PROVING %
%   B3:2/5  FE_VALVE_PROVING  "Fault Enable" %
% Rung: 19 %
% When input is enabled, a consecent change of state will be held untill "Heater OFF" or a "Fault Catch Reset" %
SOR XIC I:0.0/0 XIO B3:3/15 BST XIC B3:2/5 XIO I:0.0/5 NXB XIC B3:3/5 BND OTE B3:3/5 EOR
%   I:0.0/0  HEATER_ENABLED %
%   B3:3/15  FC_RESET %
%   B3:2/5  FE_VALVE_PROVING  "Fault Enable" %
%   I:0.0/5  VALVE_PROVING %
%   B3:3/5  FC_VALVE_PROVING  "Fault Catch" %
% Rung: 20 %
SOR XIC I:0.0/5 BST XIC I:0.0/6 NXB XIC B3:0/15 BND OTE B3:1/6 EOR
%   I:0.0/5  VALVE_PROVING %
%   I:0.0/6  HIGH_GAS_PRESSURE %
%   B3:0/15  ALARM_FLASH %
%   B3:1/6  IN_6  "High Gas Pressure" %
% Rung: 21 %
% When "Heater ON", setup input for Fault Catch and hold %
SOR XIC I:0.0/0 XIO B3:3/15 BST XIC I:0.0/6 NXB XIC B3:2/6 BND OTE B3:2/6 EOR
%   I:0.0/0  HEATER_ENABLED %
%   B3:3/15  FC_RESET %
%   I:0.0/6  HIGH_GAS_PRESSURE %
%   B3:2/6  FE_HIGH_GAS_PRES  "Fault Enable" %

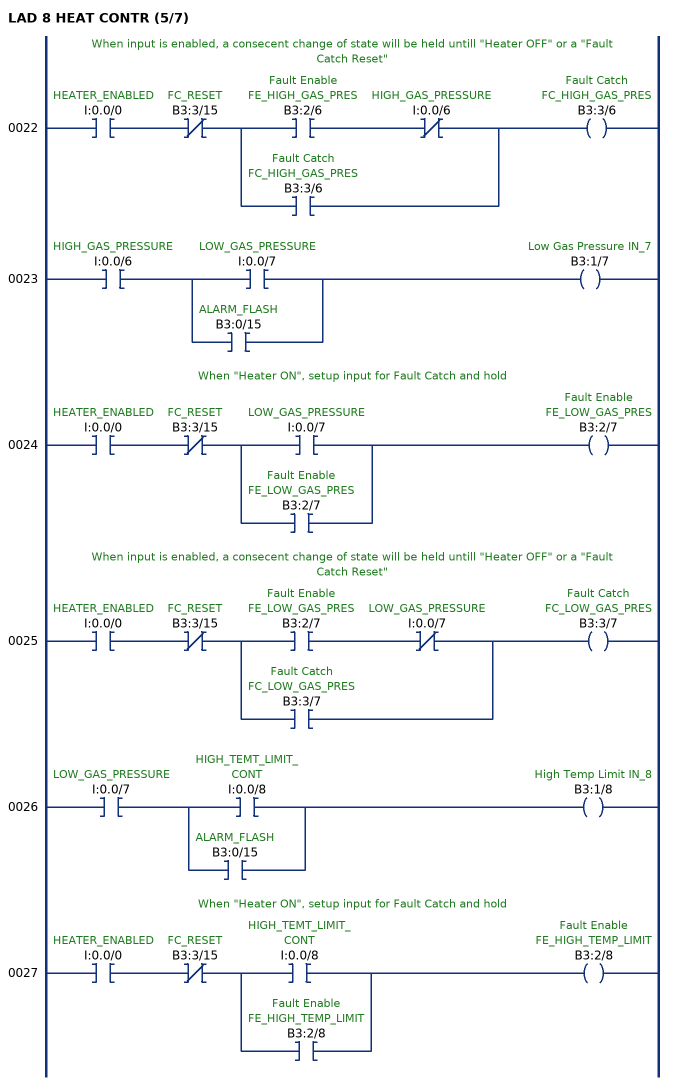
% Rung: 22 %
% When input is enabled, a consecent change of state will be held untill "Heater OFF" or a "Fault Catch Reset" %
SOR XIC I:0.0/0 XIO B3:3/15 BST XIC B3:2/6 XIO I:0.0/6 NXB XIC B3:3/6 BND OTE B3:3/6 EOR
%   I:0.0/0  HEATER_ENABLED %
%   B3:3/15  FC_RESET %
%   B3:2/6  FE_HIGH_GAS_PRES  "Fault Enable" %
%   I:0.0/6  HIGH_GAS_PRESSURE %
%   B3:3/6  FC_HIGH_GAS_PRES  "Fault Catch" %
% Rung: 23 %
SOR XIC I:0.0/6 BST XIC I:0.0/7 NXB XIC B3:0/15 BND OTE B3:1/7 EOR
%   I:0.0/6  HIGH_GAS_PRESSURE %
%   I:0.0/7  LOW_GAS_PRESSURE %
%   B3:0/15  ALARM_FLASH %
%   B3:1/7  IN_7  "Low Gas Pressure" %
% Rung: 24 %
% When "Heater ON", setup input for Fault Catch and hold %
SOR XIC I:0.0/0 XIO B3:3/15 BST XIC I:0.0/7 NXB XIC B3:2/7 BND OTE B3:2/7 EOR
%   I:0.0/0  HEATER_ENABLED %
%   B3:3/15  FC_RESET %
%   I:0.0/7  LOW_GAS_PRESSURE %
%   B3:2/7  FE_LOW_GAS_PRES  "Fault Enable" %
% Rung: 25 %
% When input is enabled, a consecent change of state will be held untill "Heater OFF" or a "Fault Catch Reset" %
SOR XIC I:0.0/0 XIO B3:3/15 BST XIC B3:2/7 XIO I:0.0/7 NXB XIC B3:3/7 BND OTE B3:3/7 EOR
%   I:0.0/0  HEATER_ENABLED %
%   B3:3/15  FC_RESET %
%   B3:2/7  FE_LOW_GAS_PRES  "Fault Enable" %
%   I:0.0/7  LOW_GAS_PRESSURE %
%   B3:3/7  FC_LOW_GAS_PRES  "Fault Catch" %
% Rung: 26 %
SOR XIC I:0.0/7 BST XIC I:0.0/8 NXB XIC B3:0/15 BND OTE B3:1/8 EOR
%   I:0.0/7  LOW_GAS_PRESSURE %
%   I:0.0/8  HIGH_TEMT_LIMIT_CONT %
%   B3:0/15  ALARM_FLASH %
%   B3:1/8  IN_8  "High Temp Limit" %
% Rung: 27 %
% When "Heater ON", setup input for Fault Catch and hold %
SOR XIC I:0.0/0 XIO B3:3/15 BST XIC I:0.0/8 NXB XIC B3:2/8 BND OTE B3:2/8 EOR
%   I:0.0/0  HEATER_ENABLED %
%   B3:3/15  FC_RESET %
%   I:0.0/8  HIGH_TEMT_LIMIT_CONT %
%   B3:2/8  FE_HIGH_TEMP_LIMIT  "Fault Enable" %

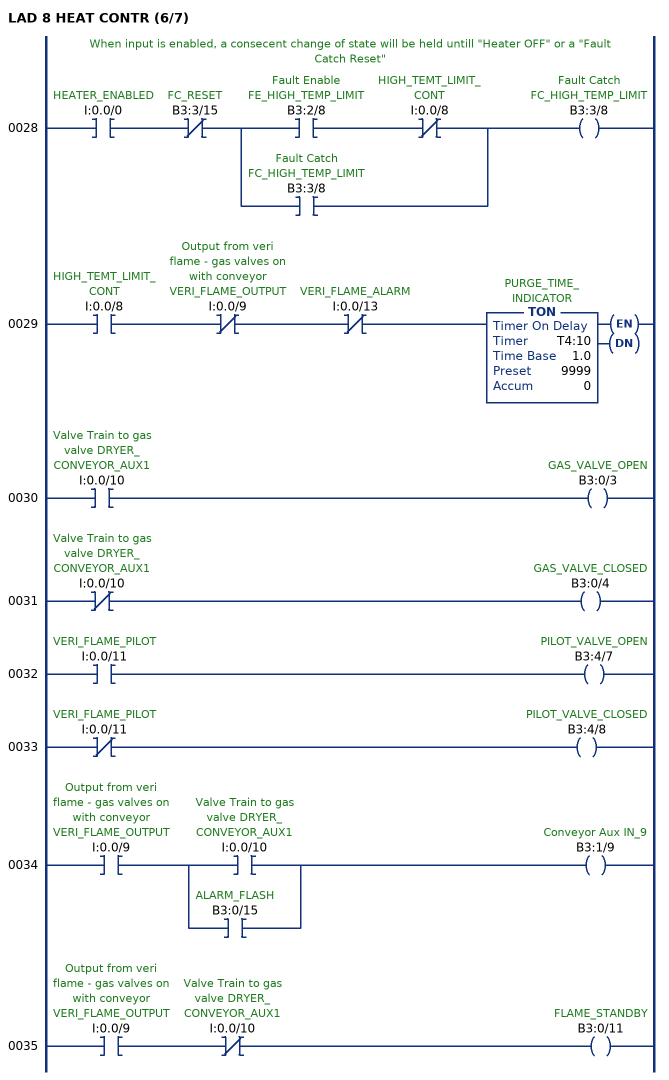
% Rung: 28 %
% When input is enabled, a consecent change of state will be held untill "Heater OFF" or a "Fault Catch Reset" %
SOR XIC I:0.0/0 XIO B3:3/15 BST XIC B3:2/8 XIO I:0.0/8 NXB XIC B3:3/8 BND OTE B3:3/8 EOR
%   I:0.0/0  HEATER_ENABLED %
%   B3:3/15  FC_RESET %
%   B3:2/8  FE_HIGH_TEMP_LIMIT  "Fault Enable" %
%   I:0.0/8  HIGH_TEMT_LIMIT_CONT %
%   B3:3/8  FC_HIGH_TEMP_LIMIT  "Fault Catch" %
% Rung: 29 %
SOR XIC I:0.0/8 XIO I:0.0/9 XIO I:0.0/13 TON T4:10 1.0 9999 0 EOR
%   I:0.0/8  HIGH_TEMT_LIMIT_CONT %
%   I:0.0/9  VERI_FLAME_OUTPUT  "Output from veri flame - gas valves on with conveyor" %
%   I:0.0/13  VERI_FLAME_ALARM %
%   T4:10  PURGE_TIME_INDICATOR %
% Rung: 30 %
SOR XIC I:0.0/10 OTE B3:0/3 EOR
%   I:0.0/10  DRYER_CONVEYOR_AUX1  "Valve Train to gas valve" %
%   B3:0/3  GAS_VALVE_OPEN %
% Rung: 31 %
SOR XIO I:0.0/10 OTE B3:0/4 EOR
%   I:0.0/10  DRYER_CONVEYOR_AUX1  "Valve Train to gas valve" %
%   B3:0/4  GAS_VALVE_CLOSED %
% Rung: 32 %
SOR XIC I:0.0/11 OTE B3:4/7 EOR
%   I:0.0/11  VERI_FLAME_PILOT %
%   B3:4/7  PILOT_VALVE_OPEN %
% Rung: 33 %
SOR XIO I:0.0/11 OTE B3:4/8 EOR
%   I:0.0/11  VERI_FLAME_PILOT %
%   B3:4/8  PILOT_VALVE_CLOSED %
% Rung: 34 %
SOR XIC I:0.0/9 BST XIC I:0.0/10 NXB XIC B3:0/15 BND OTE B3:1/9 EOR
%   I:0.0/9  VERI_FLAME_OUTPUT  "Output from veri flame - gas valves on with conveyor" %
%   I:0.0/10  DRYER_CONVEYOR_AUX1  "Valve Train to gas valve" %
%   B3:0/15  ALARM_FLASH %
%   B3:1/9  IN_9  "Conveyor Aux" %
% Rung: 35 %
SOR XIC I:0.0/9 XIO I:0.0/10 OTE B3:0/11 EOR
%   I:0.0/9  VERI_FLAME_OUTPUT  "Output from veri flame - gas valves on with conveyor" %
%   I:0.0/10  DRYER_CONVEYOR_AUX1  "Valve Train to gas valve" %
%   B3:0/11  FLAME_STANDBY %

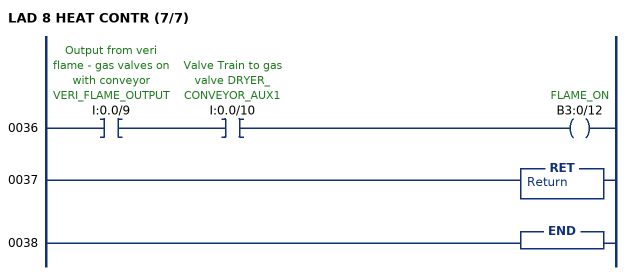
% Rung: 36 %
SOR XIC I:0.0/9 XIC I:0.0/10 OTE B3:0/12 EOR
%   I:0.0/9  VERI_FLAME_OUTPUT  "Output from veri flame - gas valves on with conveyor" %
%   I:0.0/10  DRYER_CONVEYOR_AUX1  "Valve Train to gas valve" %
%   B3:0/12  FLAME_ON %
% Rung: 37 %
SOR RET EOR
% Rung: 38 %
SOR END EOR

LADDER 9 "HOUR METER"
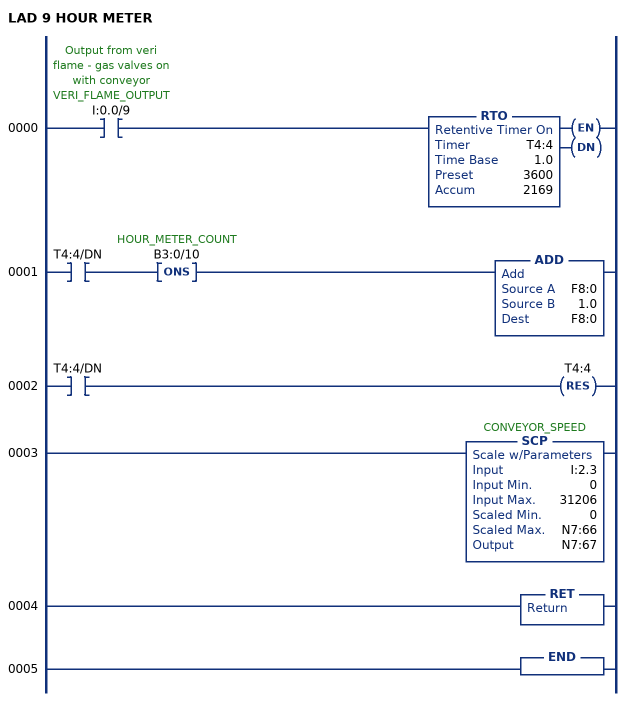
% Rung: 0 %
SOR XIC I:0.0/9 RTO T4:4 1.0 3600 2169 EOR
%   I:0.0/9  VERI_FLAME_OUTPUT  "Output from veri flame - gas valves on with conveyor" %
% Rung: 1 %
SOR XIC T4:4/DN ONS B3:0/10 ADD F8:0 1.0 F8:0 EOR
%   B3:0/10  HOUR_METER_COUNT %
% Rung: 2 %
SOR XIC T4:4/DN RES T4:4 EOR
% Rung: 3 %
SOR SCP I:2.3 0 31206 0 N7:66 N7:67 EOR
%   N7:66  CONV_SPEED_SCALLER %
%   N7:67  CONVEYOR_SPEED %
% Rung: 4 %
SOR RET EOR
% Rung: 5 %
SOR END EOR

LADDER 10 "CONV CLEAN"    % Brush Cleaning %
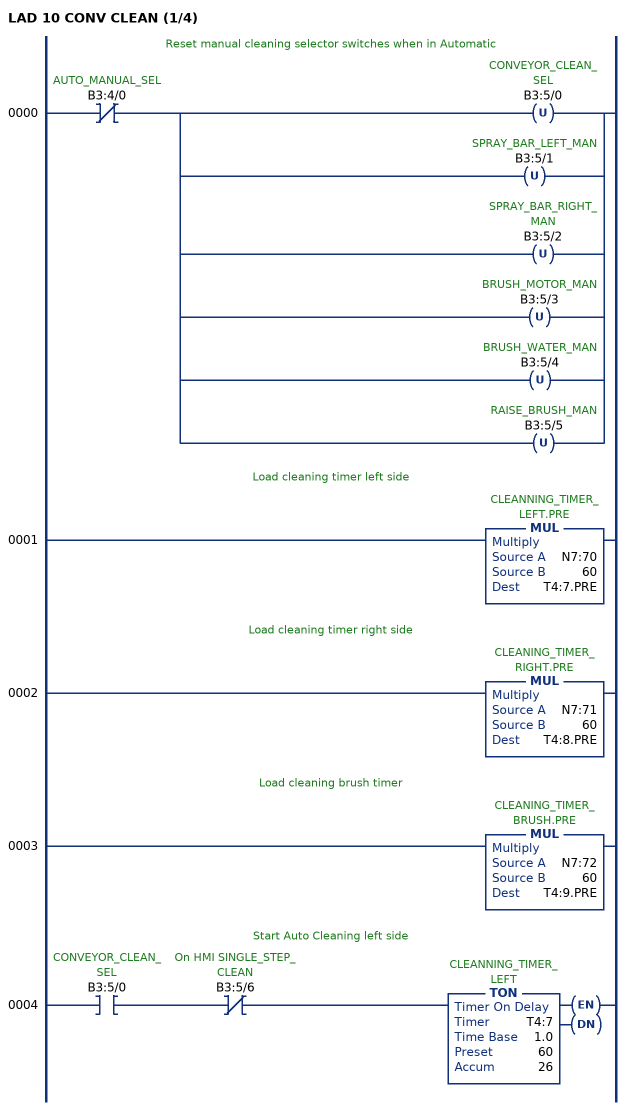
% Rung: 0 %
% Reset manual cleaning selector switches when in Automatic %
SOR XIO B3:4/0 BST OTU B3:5/0 NXB OTU B3:5/1 NXB BST OTU B3:5/2 NXB BST OTU B3:5/3 NXB BST OTU B3:5/4 NXB OTU B3:5/5 BND BND BND BND EOR
%   B3:4/0  AUTO_MANUAL_SEL %
%   B3:5/0  CONVEYOR_CLEAN_SEL %
%   B3:5/1  SPRAY_BAR_LEFT_MAN %
%   B3:5/2  SPRAY_BAR_RIGHT_MAN %
%   B3:5/3  BRUSH_MOTOR_MAN %
%   B3:5/4  BRUSH_WATER_MAN %
%   B3:5/5  RAISE_BRUSH_MAN %
% Rung: 1 %
% Load cleaning timer left side %
SOR MUL N7:70 60 T4:7.PRE EOR
%   N7:70  CLEANING_TIME_LEFT %
%   T4:7  CLEANNING_TIMER_LEFT %
% Rung: 2 %
% Load cleaning timer right side %
SOR MUL N7:71 60 T4:8.PRE EOR
%   N7:71  CLEANING_TIME_RIGHT %
%   T4:8  CLEANING_TIMER_RIGHT %
% Rung: 3 %
% Load cleaning brush timer %
SOR MUL N7:72 60 T4:9.PRE EOR
%   N7:72  CLEANING_TIME_BRUSH %
%   T4:9  CLEANING_TIMER_BRUSH %
% Rung: 4 %
% Start Auto Cleaning left side %
SOR XIC B3:5/0 XIO B3:5/6 TON T4:7 1.0 60 26 EOR
%   B3:5/0  CONVEYOR_CLEAN_SEL %
%   B3:5/6  SINGLE_STEP_CLEAN  "On HMI" %
%   T4:7  CLEANNING_TIMER_LEFT %

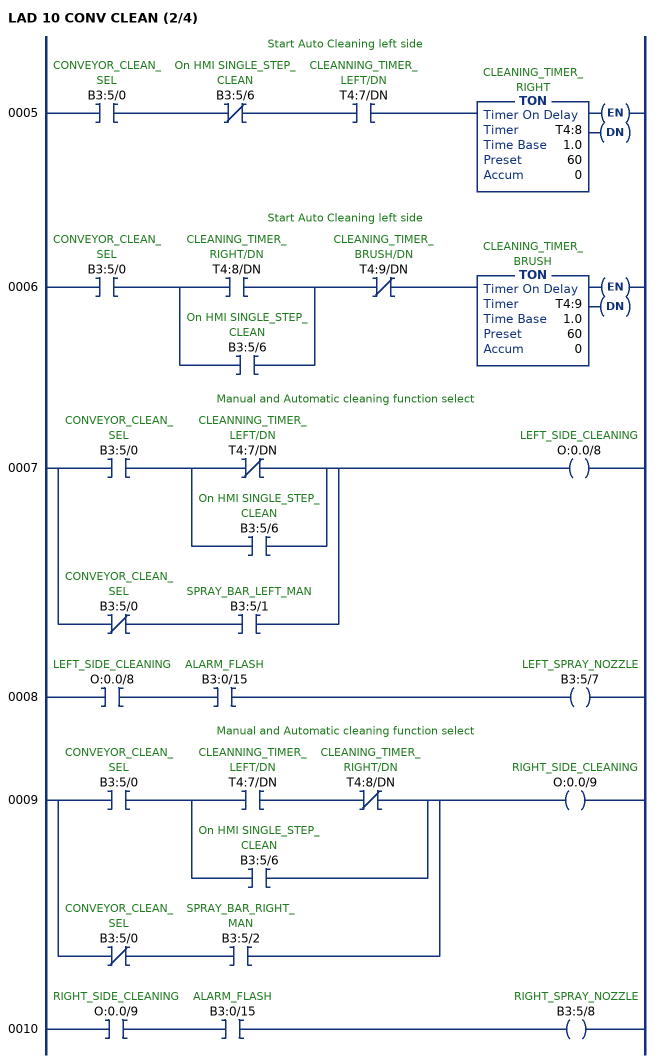
% Rung: 5 %
% Start Auto Cleaning left side %
SOR XIC B3:5/0 XIO B3:5/6 XIC T4:7/DN TON T4:8 1.0 60 0 EOR
%   B3:5/0  CONVEYOR_CLEAN_SEL %
%   B3:5/6  SINGLE_STEP_CLEAN  "On HMI" %
%   T4:7  CLEANNING_TIMER_LEFT %
%   T4:8  CLEANING_TIMER_RIGHT %
% Rung: 6 %
% Start Auto Cleaning left side %
SOR XIC B3:5/0 BST XIC T4:8/DN NXB XIC B3:5/6 BND XIO T4:9/DN TON T4:9 1.0 60 0 EOR
%   B3:5/0  CONVEYOR_CLEAN_SEL %
%   T4:8  CLEANING_TIMER_RIGHT %
%   B3:5/6  SINGLE_STEP_CLEAN  "On HMI" %
%   T4:9  CLEANING_TIMER_BRUSH %
% Rung: 7 %
% Manual and Automatic cleaning function select %
SOR BST XIC B3:5/0 BST XIO T4:7/DN NXB XIC B3:5/6 BND NXB XIO B3:5/0 XIC B3:5/1 BND OTE O:0.0/8 EOR
%   B3:5/0  CONVEYOR_CLEAN_SEL %
%   T4:7  CLEANNING_TIMER_LEFT %
%   B3:5/6  SINGLE_STEP_CLEAN  "On HMI" %
%   B3:5/1  SPRAY_BAR_LEFT_MAN %
%   O:0.0/8  LEFT_SIDE_CLEANING %
% Rung: 8 %
SOR XIC O:0.0/8 XIC B3:0/15 OTE B3:5/7 EOR
%   O:0.0/8  LEFT_SIDE_CLEANING %
%   B3:0/15  ALARM_FLASH %
%   B3:5/7  LEFT_SPRAY_NOZZLE %
% Rung: 9 %
% Manual and Automatic cleaning function select %
SOR BST XIC B3:5/0 BST XIC T4:7/DN XIO T4:8/DN NXB XIC B3:5/6 BND NXB XIO B3:5/0 XIC B3:5/2 BND OTE O:0.0/9 EOR
%   B3:5/0  CONVEYOR_CLEAN_SEL %
%   T4:7  CLEANNING_TIMER_LEFT %
%   T4:8  CLEANING_TIMER_RIGHT %
%   B3:5/6  SINGLE_STEP_CLEAN  "On HMI" %
%   B3:5/2  SPRAY_BAR_RIGHT_MAN %
%   O:0.0/9  RIGHT_SIDE_CLEANING %
% Rung: 10 %
SOR XIC O:0.0/9 XIC B3:0/15 OTE B3:5/8 EOR
%   O:0.0/9  RIGHT_SIDE_CLEANING %
%   B3:0/15  ALARM_FLASH %
%   B3:5/8  RIGHT_SPRAY_NOZZLE %

